(*
SPDX-FileCopyrightText: © 2026 Oleksandr Tiutyk <trofimich@gmail.com>
SPDX-License-Identifier: MIT
License: https://opensource.org/license/mit
*)

(*!
<summary>
Beckhoff EL2002_EX: Extended 2-channel digital output terminal with diagnostics.
</summary>
<description>
Extends EL2002 with EtherCAT Working Counter and slave state diagnostics.
When used for I/O, link located fields or their containing buffers to the matching selected PDOs.
The record is not a packed wire buffer; compiler padding is not part of the device specification.
Unlinked/default values do not prove valid I/O. The caller evaluates bus/channel validity before use.
Use one owner task per instance and externally synchronize other access; multi-field snapshots are not atomic.
Copies store data without creating hardware links. Keep borrowed field references valid while consumers are bound.
This passive record performs no validation, synchronization, configuration or protocol advancement.
WcState=TRUE means process-data exchange is invalid. State is acyclic EtherCAT/link information,
not proof of current measurement validity. Link diagnostics to the matching slave InfoData entries.
The selected PDO representation is documented by the base terminal model.
</description>
*)
TYPE EL2002_EX EXTENDS EL2002 :
STRUCT
	WcState AT %I* : BOOL;
	State AT %I* : UINT;
END_STRUCT
END_TYPE

(* stored: Version 1.1.0.1, ProductVersion 3.1.4026.18
   DUT EL2002_EX: Id {53d7c15a-469e-498f-8c28-e030ebc8e11c} *)
